// TIA Portal V21 export
FUNCTION "FC_Seguridad" : Void   // FC1, FBD
TITLE = Funcion de seguridad
{ S7_Optimized_Access := 'TRUE' }
// stored: SetENOAutomatically false
   VAR_INPUT
      "Emergency stop" : Bool;
      Start : Bool;
      Stop : Bool;
      Reset : Bool;
      "Modo auto" : Bool;
   END_VAR
   VAR_OUTPUT
      "Start Light" : Bool;
      "Reset Light" : Bool;
      "Stop Light" : Bool;
   END_VAR
BEGIN

REGION Network 1: Aviso de emergencia
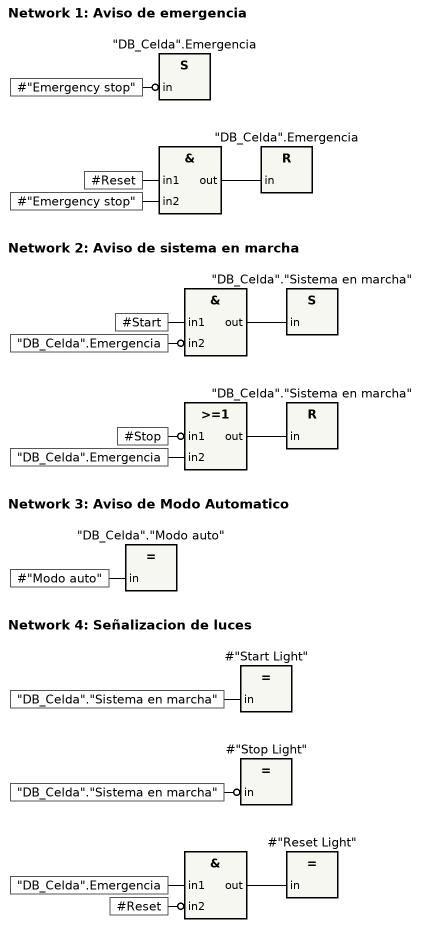
   IF NOT #"Emergency stop" THEN "DB_Celda".Emergencia := TRUE; END_IF;
   IF #Reset AND #"Emergency stop" THEN "DB_Celda".Emergencia := FALSE; END_IF;
END_REGION

REGION Network 2: Aviso de sistema en marcha
   IF #Start AND NOT "DB_Celda".Emergencia THEN "DB_Celda"."Sistema en marcha" := TRUE; END_IF;
   IF NOT #Stop OR "DB_Celda".Emergencia THEN "DB_Celda"."Sistema en marcha" := FALSE; END_IF;
END_REGION

REGION Network 3: Aviso de Modo Automatico
   "DB_Celda"."Modo auto" := #"Modo auto";
END_REGION

REGION Network 4: Señalizacion de luces
   #"Start Light" := "DB_Celda"."Sistema en marcha";
   #"Stop Light" := NOT "DB_Celda"."Sistema en marcha";
   #"Reset Light" := "DB_Celda".Emergencia AND NOT #Reset;
END_REGION
END_FUNCTION
